// Mitsubishi GX Works2 project: 2023-04-13 #1   PLC: Q03UDV
// 생산자동화기능사

// global labels: Global1
VAR_GLOBAL
  PB1 AT X0 : BOOL;
  PB2 AT X1 : BOOL;
  정지 AT X2 : BOOL;
  공급후진 AT X3 : BOOL;
  공급전진 AT X4 : BOOL;
  가공후진 AT X5 : BOOL;
  가공전진 AT X6 : BOOL;
  송출후진 AT X7 : BOOL;
  송출전진 AT X8 : BOOL;
  배출후진 AT X9 : BOOL;
  배출전진 AT X0A : BOOL;
  매거진 AT X0B : BOOL;
  가공센서 AT X0C : BOOL;
  송출센서 AT X0D : BOOL;
  비금속센서 AT X0E : BOOL;
  금속센서 AT X0F : BOOL;
  적색 AT Y20 : BOOL;
  황색 AT Y21 : BOOL;
  녹색 AT Y22 : BOOL;
  공급1 AT Y23 : BOOL;
  공급2 AT Y24 : BOOL;
  가공 AT Y25 : BOOL;
  드릴 AT Y26 : BOOL;
  송출 AT Y27 : BOOL;
  배출 AT Y28 : BOOL;
  컨베이어 AT Y29 : BOOL;
END_VAR

PROGRAM 기본동작
VAR
  STATE : INT;
END_VAR
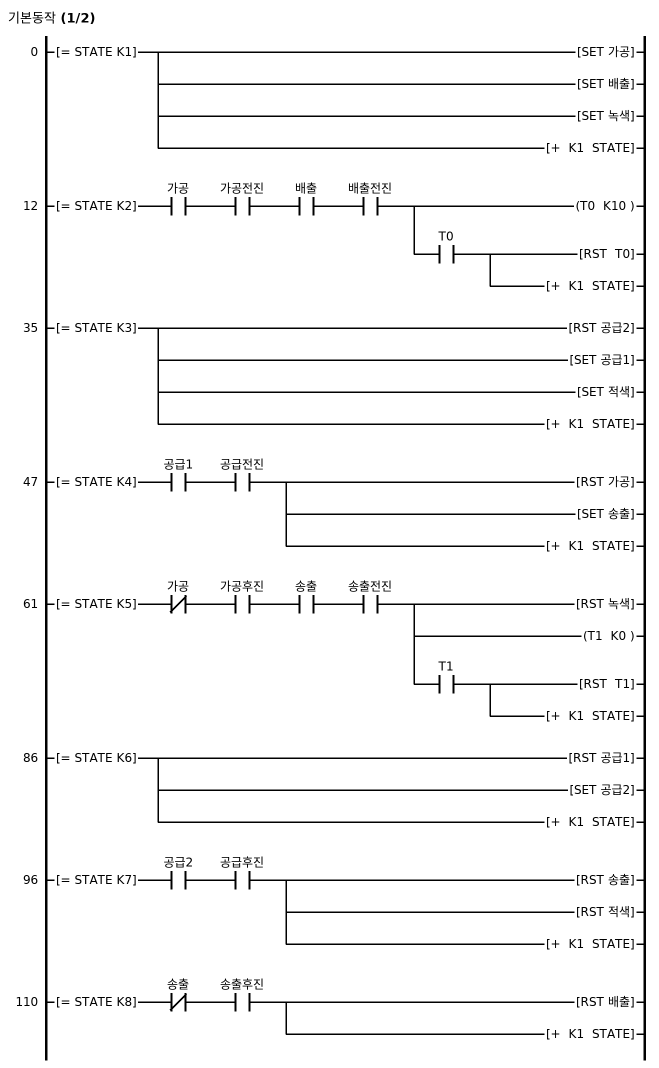
0     LD=     STATE K1
      SET     가공
      SET     배출
      SET     녹색
      +       K1 STATE
12    LD=     STATE K2
      AND     가공
      AND     가공전진
      AND     배출
      AND     배출전진
      OUT     T0 K10
      AND     T0
      RST     T0
      +       K1 STATE
35    LD=     STATE K3
      RST     공급2
      SET     공급1
      SET     적색
      +       K1 STATE
47    LD=     STATE K4
      AND     공급1
      AND     공급전진
      RST     가공
      SET     송출
      +       K1 STATE
61    LD=     STATE K5
      ANI     가공
      AND     가공후진
      AND     송출
      AND     송출전진
      RST     녹색
      OUT     T1 K0
      AND     T1
      RST     T1
      +       K1 STATE
86    LD=     STATE K6
      RST     공급1
      SET     공급2
      +       K1 STATE
96    LD=     STATE K7
      AND     공급2
      AND     공급후진
      RST     송출
      RST     적색
      +       K1 STATE
110   LD=     STATE K8
      ANI     송출
      AND     송출후진
      RST     배출
      +       K1 STATE
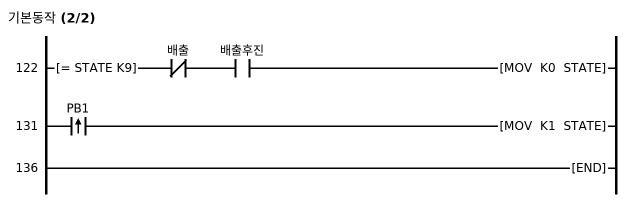
122   LD=     STATE K9
      ANI     배출
      AND     배출후진
      MOV     K0 STATE
131   LDP     PB1
      MOV     K1 STATE
136   END
END_PROGRAM

PROGRAM 응용동작1
VAR
  STATE : INT;
END_VAR
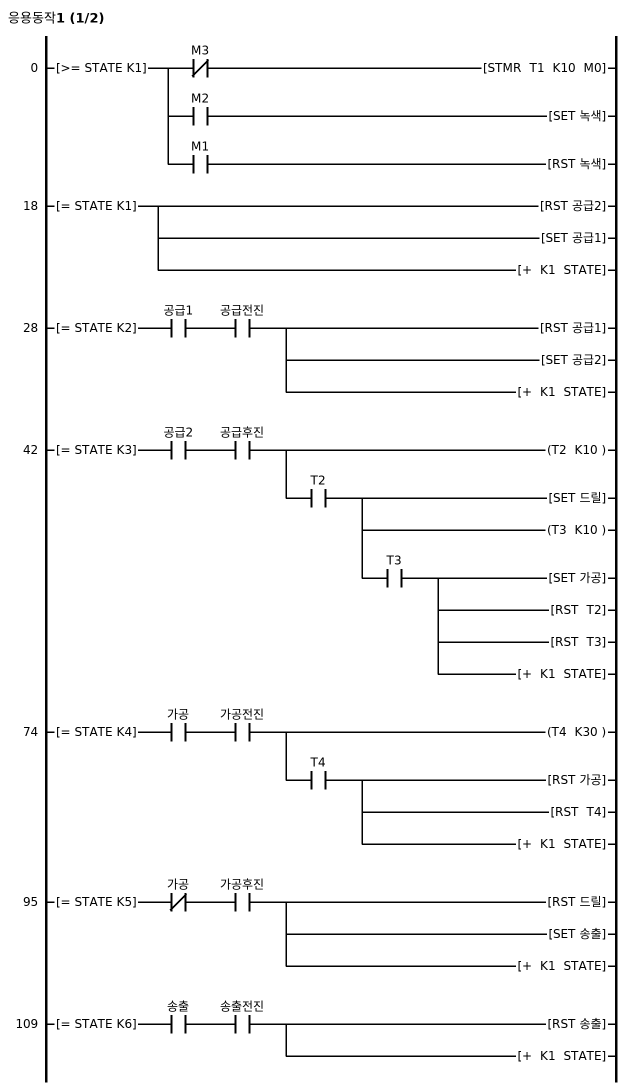
0     LD>=    STATE K1
      MPS
      ANI     M3
      STMR    T1 K10 M0
      MRD
      AND     M2
      SET     녹색
      MPP
      AND     M1
      RST     녹색
18    LD=     STATE K1
      RST     공급2
      SET     공급1
      +       K1 STATE
28    LD=     STATE K2
      AND     공급1
      AND     공급전진
      RST     공급1
      SET     공급2
      +       K1 STATE
42    LD=     STATE K3
      AND     공급2
      AND     공급후진
      OUT     T2 K10
      AND     T2
      SET     드릴
      OUT     T3 K10
      AND     T3
      SET     가공
      RST     T2
      RST     T3
      +       K1 STATE
74    LD=     STATE K4
      AND     가공
      AND     가공전진
      OUT     T4 K30
      AND     T4
      RST     가공
      RST     T4
      +       K1 STATE
95    LD=     STATE K5
      ANI     가공
      AND     가공후진
      RST     드릴
      SET     송출
      +       K1 STATE
109   LD=     STATE K6
      AND     송출
      AND     송출전진
      RST     송출
      +       K1 STATE
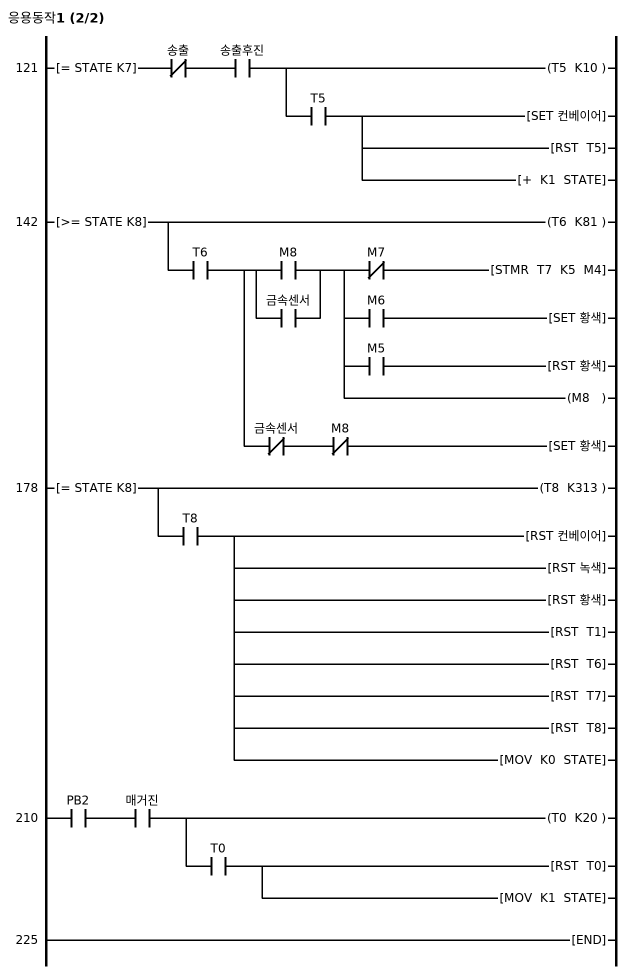
121   LD=     STATE K7
      ANI     송출
      AND     송출후진
      OUT     T5 K10
      AND     T5
      SET     컨베이어
      RST     T5
      +       K1 STATE
142   LD>=    STATE K8
      OUT     T6 K81
      AND     T6
      MPS
      LD      M8
      OR      금속센서
      ANB
      MPS
      ANI     M7
      STMR    T7 K5 M4
      MRD
      AND     M6
      SET     황색
      MRD
      AND     M5
      RST     황색
      MPP
      OUT     M8
      MPP
      ANI     금속센서
      ANI     M8
      SET     황색
178   LD=     STATE K8
      OUT     T8 K313
      AND     T8
      RST     컨베이어
      RST     녹색
      RST     황색
      RST     T1
      RST     T6
      RST     T7
      RST     T8
      MOV     K0 STATE
210   LD      PB2
      AND     매거진
      OUT     T0 K20
      AND     T0
      RST     T0
      MOV     K1 STATE
225   END
END_PROGRAM
